{attribute 'qualified_only'}
{attribute 'strict'}
TYPE E_MR1L0_CoatingStates :
(
    Unknown := 0,
    L0B4C := 1,
    L0Ni := 2,
    L1B4C := 3,
    L1Ni := 4
) UINT;
END_TYPE

(* stored: Version 1.1.0.1, ProductVersion 3.1.4022.18
   DUT E_MR1L0_CoatingStates: Id {47798397-c26e-413b-9427-6a3684e9f159} *)
